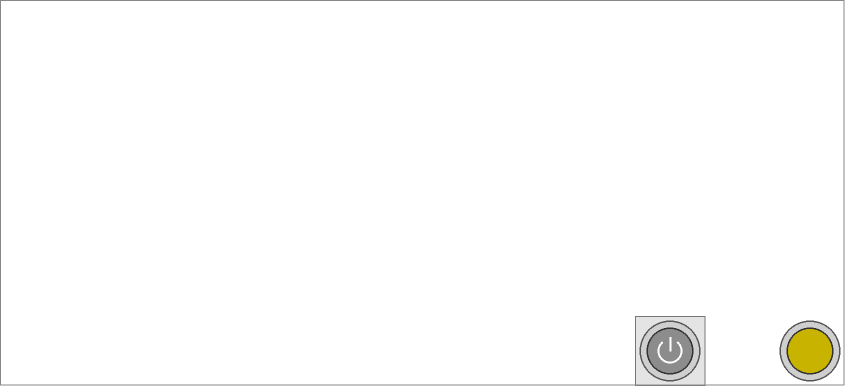
VISUALIZATION Visu  // 845x386
    Lamp1 (775,316 70x70), variable: MAIN.Q01, style: Lamp-Lamp1-Yellow
    PowerSwitch (635,316 70x70), variable: MAIN.S01, behaviour: TOGGLE, style: Switch-PowerSwitch-Gray
END_VISUALIZATION

(* stored: Version 1.1.0.1, ProductVersion 3.1.4024.12
   Visu Visu: Id {3902bc4a-b3aa-4a56-bb5b-ebca5a4be039} *)
